(* LS Electric XG5000 project: 20230514_PLC_01 *)
(* PLC LSPLC *)

PROGRAM NewProgram (* task: 스캔 프로그램 *)
VAR
    결과 : INT;
    결과_R : REAL;
    램프1 : BOOL;
    램프2 : BOOL;
    램프3 : BOOL;
    램프4 : BOOL;
    램프4_1 : BOOL;
    램프4_2 : BOOL;
    램프4_3 : BOOL;
    셋코일1 : BOOL;
    숫자1 : INT;
    숫자1_R : REAL;
    스위치1 : BOOL;
    스위치2 : BOOL;
    스위치3 : BOOL;
    스위치4 : BOOL;
    음변환 : BOOL;
    음변환_램프 : BOOL;
    정지 : BOOL;
END_VAR
VAR
    _e1 : R_TRIG;
    _e2 : F_TRIG;
    _e3 : R_TRIG;
    _e4 : R_TRIG;
    _e5 : R_TRIG;
    _e6 : R_TRIG;
END_VAR

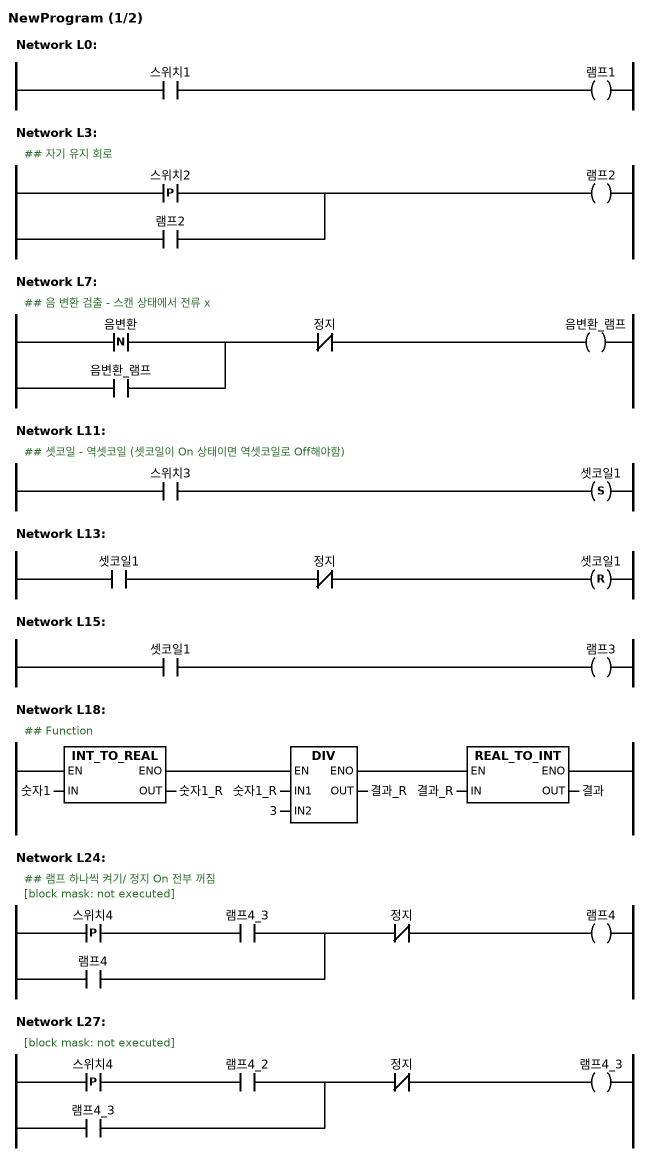
(* Rung L0 *)
램프1 := 스위치1;
(* ## 자기 유지 회로 *)
(* Rung L3 *)
_e1(CLK := 스위치2);
램프2 := _e1.Q OR 램프2;
(* ## 음 변환 검출 - 스캔 상태에서 전류 x *)
(* Rung L7 *)
_e2(CLK := 음변환);
음변환_램프 := (_e2.Q OR 음변환_램프) AND NOT 정지;
(* ## 셋코일 - 역셋코일 (셋코일이 On 상태이면 역셋코일로 Off해야함) *)
(* Rung L11 *)
IF 스위치3 THEN 셋코일1 := TRUE; END_IF;
(* Rung L13 *)
IF 셋코일1 AND NOT 정지 THEN 셋코일1 := FALSE; END_IF;
(* Rung L15 *)
램프3 := 셋코일1;
(* ## Function *)
(* Rung L18 *)
숫자1_R := INT_TO_REAL(숫자1);
결과_R := 숫자1_R / 3;
결과 := REAL_TO_INT(결과_R);
(* ## 램프 하나씩 켜기/ 정지 On 전부 꺼짐 *)
(* Rung L24 is block-masked: not executed *)
// _e3(CLK := 스위치4);
// 램프4 := ((_e3.Q AND 램프4_3) OR 램프4) AND NOT 정지;
(* Rung L27 is block-masked: not executed *)
// _e4(CLK := 스위치4);
// 램프4_3 := ((_e4.Q AND 램프4_2) OR 램프4_3) AND NOT 정지;

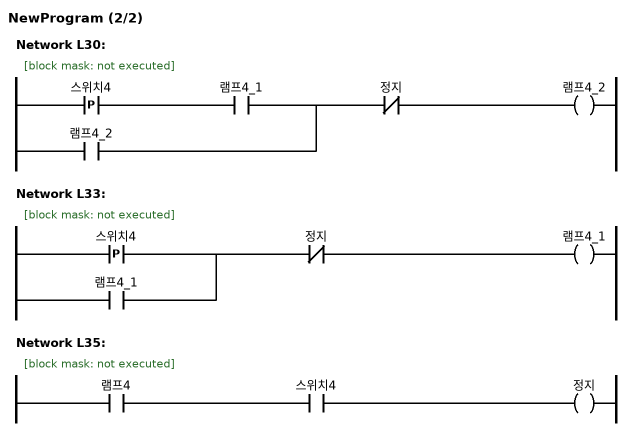
(* Rung L30 is block-masked: not executed *)
// _e5(CLK := 스위치4);
// 램프4_2 := ((_e5.Q AND 램프4_1) OR 램프4_2) AND NOT 정지;
(* Rung L33 is block-masked: not executed *)
// _e6(CLK := 스위치4);
// 램프4_1 := (_e6.Q OR 램프4_1) AND NOT 정지;
(* Rung L35 is block-masked: not executed *)
// 정지 := 램프4 AND 스위치4;
END_PROGRAM